TYPE ST_ModuleRuntimeConfig :
STRUCT
	Enabled : BOOL;
	Valid : BOOL;
	ModuleId : UDINT;
	ModuleType : STRING(16);
	AdsPort : UINT;
	Revision : UDINT;
	VariableCount : UINT;
	VariableList : ARRAY[1..Param_Config.MaxModuleVariable] OF ST_ConfigVariableInfo;
	AlarmCount : UINT;
	AlarmList : ARRAY[1..Param_Config.MaxConfiguredAlarmsPerModule] OF ST_ConfigAlarmInfo;
END_STRUCT
END_TYPE

(* stored: Version 1.1.0.1, ProductVersion 3.1.4026.18
   DUT ST_ModuleRuntimeConfig: Id {a3b51235-1e4c-4a0d-841f-c1f732d4a3b5} *)
